{attribute 'TcGenerated'}
{attribute 'no-analysis'}
{attribute 'linkalways'}
// This function has been automatically generated from the project information.
VAR_GLOBAL CONSTANT
	{attribute 'const_non_replaced'}
	stLibVersion_TwinCAT_Open_Framework_Tasks : ST_LibVersion := (iMajor := 1, iMinor := 0, iBuild := 13, iRevision := 0, nFlags := 0, sVersion := '1.0.13.0');
END_VAR

(* stored: Version 1.1.0.1
   GVL Global_Version: Id {49c87b01-f23e-432f-a86c-51f154886757} *)
